PROGRAM MAIN
VAR
END_VAR

END_PROGRAM

(* stored: Version 1.1.0.1
   POU MAIN: Id {539be4ca-25cc-43dd-904f-f047e8f2e8d2} *)
